TYPE DUT_SilownikParametry :
STRUCT
	rCzasNaPrace							: REAL := 5000;
	rCzasNaPowrot							: REAL := 5000;
END_STRUCT
END_TYPE

(* stored: Version 1.1.0.1, ProductVersion 3.1.4024.11
   DUT DUT_SilownikParametry: Id {19b93c4e-c509-4ba3-a0d0-5e842466ad5d} *)
